// TIA Portal V18 export
DATA_BLOCK "_ML2_modeDB"   // DB12
VERSION : 0.1
// stored: AutoNumber true, DBAccessibleFromOPCUA true, InstanceOfName _ML2_mode, InstanceOfType FB
"_ML2_mode"
   // VAR_IN_OUT
   //    xSoftSTOP : Bool;
   //    yExecuteAll : Bool;
   //    yTeam_unison : Bool;
   //    yOVERRIDE : Bool;
   // END_VAR
BEGIN
END_DATA_BLOCK
